INTERFACE I_Logger EXTENDS I_Object

METHOD PUBLIC M_Log
VAR_INPUT
	Message:			STRING(255);
END_VAR
END_METHOD

END_INTERFACE

(* stored: Version 1.1.0.1
   Itf I_Logger: Id {1a1f5bf4-6529-4849-9bae-5eab010a432b}
   Method M_Log: Id {9bc8e32d-5fed-4962-a72b-a42bbceea32e} *)
